FUNCTION_BLOCK FB_DataToNovRam
VAR_INPUT
	bExecute:BOOL;
	
	savedData:ST_AlarmInfo_DB_save;
END_VAR
VAR_OUTPUT
	bResult:BOOL;
END_VAR
VAR
	
END_VAR
VAR_IN_OUT
END_VAR

METHOD M_AlarmHistory : BOOL
VAR_INPUT
	addData:ST_AlarmInfo_DB_save;
END_VAR
VAR
	i:UDINT;
END_VAR
IF GVL.NovRamData.NovRam_Status.RowDataLocked[GVL.NovRamData.NovRam_Status.nowRowIndex]=FALSE THEN//writable
	
	//write data
	GVL.NovRamData.AlarmHistory[GVL.NovRamData.NovRam_Status.nowRowIndex][GVL.NovRamData.NovRam_Status.writenIndex]:=addData;
	
	GVL.NovRamData.NovRam_Status.writenIndex:=GVL.NovRamData.NovRam_Status.writenIndex+1;
	
	//Check if Full
	IF GVL.NovRamData.NovRam_Status.writenIndex >= (GVL.AlarmHistory_ArrayLength - 1) THEN
		//Set Row Lock
		GVL.NovRamData.NovRam_Status.RowDataLocked[GVL.NovRamData.NovRam_Status.nowRowIndex]:=TRUE;
		
		//Reset Row and writenIndex
		GVL.NovRamData.NovRam_Status.nowRowIndex:=(GVL.NovRamData.NovRam_Status.nowRowIndex+1)MOD GVL.NovRamBufferRatio;
		GVL.NovRamData.NovRam_Status.writenIndex:=0;
	END_IF
	
	M_AlarmHistory:=TRUE;
ELSE
	M_AlarmHistory:=FALSE;
END_IF
END_METHOD

END_FUNCTION_BLOCK

(* stored: Version 1.1.0.1, ProductVersion 3.1.4024.11
   POU FB_DataToNovRam: Id {76f3141b-7a21-4959-afa9-90d9594b687d}, SpecialFunc None
   Method M_AlarmHistory: Id {aac47326-eba1-4863-89c8-9d8cb955d250} *)
